{attribute 'enable_dynamic_creation'}
TYPE ST_HASHSET_BUCKET_NODE :
STRUCT
	Data : T_Generic;
	pNext : POINTER TO ST_HASHSET_BUCKET_NODE;
END_STRUCT
END_TYPE

(* stored: Version 1.1.0.1
   DUT ST_HASHSET_BUCKET_NODE: Id {954d4eca-b9eb-03bb-2c08-1fe3468a4383} *)
